FUNCTION_BLOCK Proxy (* Proxy Function Block Type *)
  (* Standard: 61499-1 *)
  (* Version 0.1, 2003-12-05, JHC, Rockwell Automation, Renamed from NEWPROXY. *)
  (* Version 0.0, 2003-02-05, JHC, Rockwell Automation, Copied/Modified from IB4 example. *)
  (* Compiler header: package fb.rt.template; *)
  (* Compiler classdef: public class NEWPROXY extends FBDNProxy *)
  (* Compiler Java IBM Jikes 1.06 *)
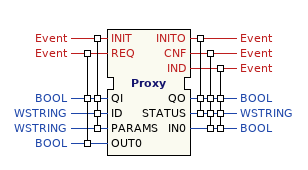
  EVENT_INPUT
    INIT WITH QI, ID, PARAMS; (* Service Initialization *)
    REQ WITH QI, OUT0; (* Data Write/Read Request *)
  END_EVENT
  EVENT_OUTPUT
    INITO WITH QO, STATUS; (* Initialization Confirm *)
    CNF WITH QO, STATUS, IN0; (* Data Arrives *)
    IND WITH QO, STATUS, IN0; (* Data Changed *)
  END_EVENT
  VAR_INPUT
    QI : BOOL; (* Event Input Qualifier *)
    ID : WSTRING; (* DNet Address *)
    PARAMS : WSTRING; (* Service Parameters *)
    OUT0 : BOOL; (* Output to device *)
  END_VAR
  VAR_OUTPUT
    QO : BOOL; (* Event Output Qualifier *)
    STATUS : WSTRING; (* Service Status *)
    IN0 : BOOL; (* Input from Device *)
  END_VAR
  SERVICE APPLICATION/resource
    SEQUENCE normal_establishment
      APPLICATION.INIT+(ID,PARAMS) -> resource.initialize(ID,PARAMS) -> APPLICATION.INITO+();
    END_SEQUENCE
    SEQUENCE unsuccessful_establishment
      APPLICATION.INIT+(ID,PARAMS) -> resource.initialize(ID,PARAMS) -> APPLICATION.INITO-(STATUS);
    END_SEQUENCE
    SEQUENCE io_no_input_change
      APPLICATION.REQ+(OUT0) -> resource.request(OUT0) -> APPLICATION.CNF+(IN0);
    END_SEQUENCE
    SEQUENCE read_data_changed
      APPLICATION.REQ+(OUT0) -> resource.request(OUT0) -> APPLICATION.CNF+(IN0,IN1,IN2,IN3) -> APPLICATION.IND+(IN0,IN1,IN2,IN3);
    END_SEQUENCE
    SEQUENCE request_inhibited
      APPLICATION.REQ-() -> APPLICATION.CNF-(STATUS);
    END_SEQUENCE
    SEQUENCE request_error
      APPLICATION.REQ+(OUT0) -> resource.request(OUT0) -> APPLICATION.CNF-(STATUS);
    END_SEQUENCE
    SEQUENCE error_notification
      resource.error() -> APPLICATION.CNF-(STATUS);
    END_SEQUENCE
    SEQUENCE application_initiated_termination
      APPLICATION.INIT-() -> resource.terminate() -> APPLICATION.INITO-(STATUS);
    END_SEQUENCE
    SEQUENCE resource_initiated_termination
      resource.terminated() -> APPLICATION.INITO-(STATUS);
    END_SEQUENCE
  END_SERVICE
END_FUNCTION_BLOCK
